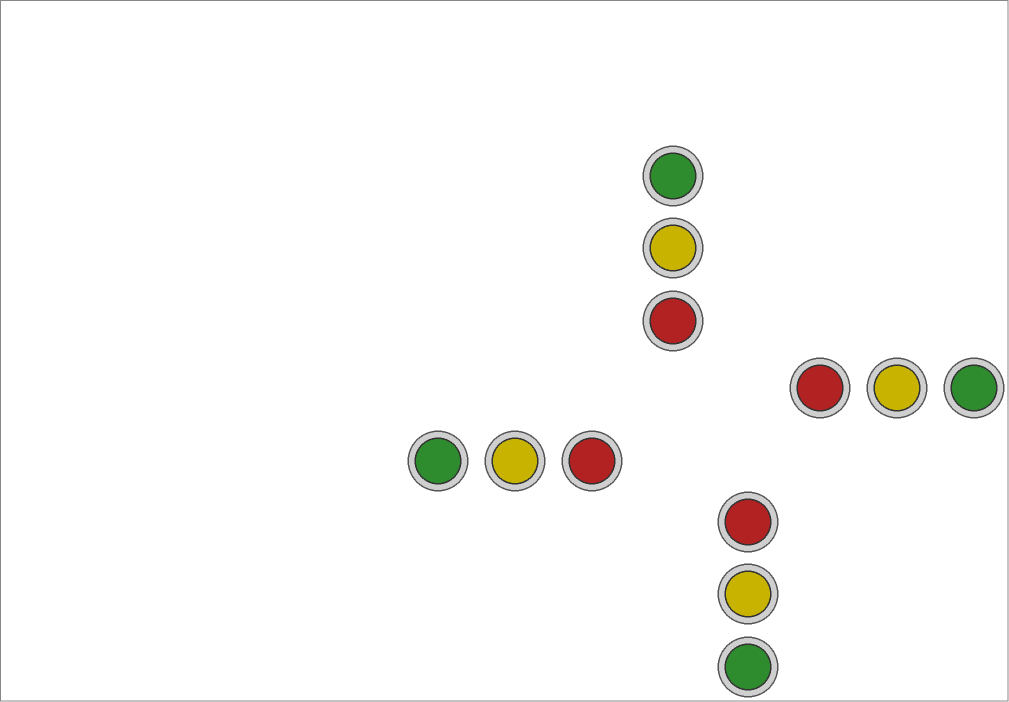
VISUALIZATION Visu  // 1009x702
    Group (403,426 224x70)
        Lamp1 (154,0 70x70), variable: MAIN.b_rood_h, style: Lamp-Lamp1-Red
        Lamp1 (77,0 70x70), variable: MAIN.b_oranje_h, style: Lamp-Lamp1-Yellow
        Lamp1 (0,0 70x70), variable: MAIN.b_groen_h, style: Lamp-Lamp1-Green
    Group (785,353 224x70)
        Lamp1 (154,0 70x70), variable: MAIN.b_groen_h, style: Lamp-Lamp1-Green
        Lamp1 (77,0 70x70), variable: MAIN.b_oranje_h, style: Lamp-Lamp1-Yellow
        Lamp1 (0,0 70x70), variable: MAIN.b_rood_h, style: Lamp-Lamp1-Red
    Group (713,487 70x215)
        Lamp1 (0,0 70x70), variable: MAIN.b_rood_v, style: Lamp-Lamp1-Red
        Lamp1 (0,72 70x70), variable: MAIN.b_oranje_v, style: Lamp-Lamp1-Yellow
        Lamp1 (0,145 70x70), variable: MAIN.b_groen_v, style: Lamp-Lamp1-Green
    Group (638,141 70x215)
        Lamp1 (0,0 70x70), variable: MAIN.b_groen_v, style: Lamp-Lamp1-Green
        Lamp1 (0,72 70x70), variable: MAIN.b_oranje_v, style: Lamp-Lamp1-Yellow
        Lamp1 (0,145 70x70), variable: MAIN.b_rood_v, style: Lamp-Lamp1-Red
END_VISUALIZATION

(* stored: Version 1.1.0.1, ProductVersion 3.1.4024.12
   Visu Visu: Id {54a6e84d-8295-4145-974e-4ad795072c4d} *)
